	rFlawWaterAfterAlcaliSet:=	arFlawWaterAfterAlcaliSet[3, wChosenRecipeLine3],
	rFlawWaterAfterAccidSet:=	arFlawWaterAfterAccidSet[3, wChosenRecipeLine3],
	rWaterAfterSterilFlaw:=	arWaterAfterSterilFlaw[3, wChosenRecipeLine3],
	rWaterAfterSterilConc:=	arWaterAfterSterilConc[3, wChosenRecipeLine3],
	rFlawWaterAfterAlcaliSet:=	arFlawWaterAfterAlcaliSet[3, wChosenRecipeLine3],
	rFlawWaterAfterAccidSet:=	arFlawWaterAfterAccidSet[3, wChosenRecipeLine3],
	wUsedWaterLevelOK:= wUsedWaterLevelOK,
	wUsedWaterLevelNotOK:= wUsedWaterLevelNotOK,
	wBackTget:= Heater_BackTget_3,
	xPause:= xPauseWashingLine3,
	xVoutOn:= xState_V311,
	xV_NotshortcutOn:= xState_V310,
	xV_UsedWaterInOn:= xState_V308,
	xV_AlkaliInOn:= xState_V306,
	xV_AccidInOn:= xState_V307,
	xV_WaterOutOn:= xState_V301,
	xV_UsedWaterOutOn:= xState_V302,
	xV_AlkaliOutOn:= xState_V304,
	xV_AccidOutOn:= xState_V303,
	xV_CycleOn:= xState_V305,
	xPumpOn:= Pump_OnAuto_3,
	rConcentration:= Conc_Line3,
	(*xAccidIsGoing:=xAccidIsGoing3,*)
	xFeedbackSwitch:= DI_FeedBackSwitchLine3,
	rWaterAfterSterilT:=arWaterAfterSterilT[3, wChosenRecipeLine3],
	wRecipeTimeRinse:= arWaterTime[3, wChosenRecipeLine3],
	wRecipeTimeAlcali:= arAlkaliTime[3, wChosenRecipeLine3],
	wRecipeTimeAccid:= arAccidTime[3, wChosenRecipeLine3],
	wAfterRinseConcAlk:= (*wAfterRinseConcAlk*)rConcSolutionStopoperationAlk,
	wAfterRinseConcAcc:= (*wAfterRinseConcAcc*)rConcSolutionStopoperationAcc,
	wAfterAlkWaterTime:= arAfterAlkaliWaterTime[3, wChosenRecipeLine3],
	wAfterAccWaterTime:= arAfterAccidWaterTime[3, wChosenRecipeLine3],
	rTwaterSet:= arTwaterSet[3, wChosenRecipeLine3],
	rTalcaliSet:= arTalkaliSet[3, wChosenRecipeLine3],
	rTaccidSet:= arTaccidSet[3, wChosenRecipeLine3],
	rConcAlcaliSet:= (*arConcAlkaliSet[3, wChosenRecipeLine3]*)rConcSolutionStartOperationAlk,
	rConcAccidSet:= (*arConcAccidSet[3, wChosenRecipeLine3]*)rConcSolutionStartOperationAcc,
	rFlawAlcaliSet:= arFlawAlkaliSet[3, wChosenRecipeLine3],
	rFlawWaterSet:= arFlawWaterSet[3, wChosenRecipeLine3],
	rFlawAccidSet:= arFlawAccidSet[3, wChosenRecipeLine3],
	wTsteril:= arTsterilSet[3, wChosenRecipeLine3],
	wFlawSteril:= arFlawSterilSet[3, wChosenRecipeLine3],
	rConcSteril:= arConcSterilSet[3, wChosenRecipeLine3],
	wSterilTime:= arSterilTime[3, wChosenRecipeLine3],
	wCountOfOperations:= 7,
	xStart:= xStartWashingLine3,
	xVout:= OnAuto_V311,
	xV_Notshortcut:= OnAuto_V310,
	xV_UsedWaterIn:= OnAuto_V308,
	xV_AlkaliIn:= OnAuto_V306,
	xV_AccidIn:= OnAuto_V307,
	xV_WaterOut:= OnAuto_V301,
	xV_UsedWaterOut:= OnAuto_V302,
	xV_AlkaliOut:= OnAuto_V304,
	xV_AccidOut:= OnAuto_V303,
	xV_Cycle:= OnAuto_V305,
	xV_Drainage:= OnAuto_V309,
	xPump:= Pump_OnAuto_3,
	xHeaterPower:= Heater_AutoSetT_3,
	xResetErrors:= xResetAlmAll,
	xPA:= PA_OnAuto_3,
	rToutSet:= Heater_AutoSetT_3,
	rFlawOutSet:= Pump_FlawAutoSet_3,
	xDone:=xWashingDone_Line3,
	State=> wWashingStateLine3,
	PauseState=>(* wWashingPauseStateLine3*),
	wTimePassed=> wWashingTimePassed3,
	wTimeOperationSet=> wWashingOperTimeSet3,
	wError=> wWashingErr_3);
END_IF
END_PROGRAM

(* POU Process/Washing/prWashingLine4, ST *)
PROGRAM prWashingLine4
VAR
	WashingProcess4:	fbWashingProcess;
	xResetErrors: BOOL;
END_VAR
IF wDissolvingStateLine4 = 0 THEN
WashingProcess4(
	xReady:= (*xReadyForWashing AND*) wDissolvingStateLine4 = 0,
	arOperations:= arOperations,
	rWaterLevel:= CleanWaterLevel,
	rUsedWaterLevel:= UsedWaterLevel,
	rAccidLevel:= AccidLevel,
	rAlkaliLevel:= AlkaliLevel,
	wConcPumpTime:=arConcPumpTimeSteril[4, wChosenRecipeLine4],
	wConcMessureTime:= rConcCheckTime,
	arOperations2x:=arOperations2x,
	arOperations3x:=arOperations3x,
	wChosenRecipeLine:=wChosenRecipeLine4,
	wLine:=4,
	rConcOfClkaliInTank:=rDissolAlkaliConcSet,
	rConcOfAccidInTank:=rDissolAccidConcSet,

	xPumpNorm:=Pump_InvNorm_4,

	rWaterAfterSterilTime:=arWaterAfterSterilTime[4, wChosenRecipeLine4],
	wTafterAlkaliWater:=arTafterAlkaliWater[4, wChosenRecipeLine4],
	wTafterAccidWater:=arTafterAccidWater[4, wChosenRecipeLine4],

	rFlawWaterAfterAlcaliSet:=	arFlawWaterAfterAlcaliSet[4, wChosenRecipeLine4],
	rFlawWaterAfterAccidSet:=	arFlawWaterAfterAccidSet[4, wChosenRecipeLine4],
	rWaterAfterSterilFlaw:=	arWaterAfterSterilFlaw[4, wChosenRecipeLine4],
	rWaterAfterSterilConc:=	arWaterAfterSterilConc[4, wChosenRecipeLine4],
	rFlawWaterAfterAlcaliSet:=	arFlawWaterAfterAlcaliSet[4, wChosenRecipeLine4],
	rFlawWaterAfterAccidSet:=	arFlawWaterAfterAccidSet[4, wChosenRecipeLine4],
	wUsedWaterLevelOK:= wUsedWaterLevelOK,
	wUsedWaterLevelNotOK:= wUsedWaterLevelNotOK,
	wBackTget:= Heater_BackTget_4,
	xPause:= xPauseWashingLine4,
	xVoutOn:= xState_V411,
	xV_NotshortcutOn:= xState_V410,
	xV_UsedWaterInOn:= xState_V408,
	xV_AlkaliInOn:= xState_V406,
	xV_AccidInOn:= xState_V407,
	xV_WaterOutOn:= xState_V401,
	xV_UsedWaterOutOn:= xState_V402,
	xV_AlkaliOutOn:= xState_V404,
	xV_AccidOutOn:= xState_V403,
	xV_CycleOn:= xState_V405,
	xPumpOn:= Pump_OnAuto_4,
	rConcentration:= Conc_Line4,
	(*xAccidIsGoing:=xAccidIsGoing4,*)
	xFeedbackSwitch:= DI_FeedBackSwitchLine4,
	rWaterAfterSterilT:=arWaterAfterSterilT[4, wChosenRecipeLine4],
	wRecipeTimeRinse:= arWaterTime[4, wChosenRecipeLine4],
	wRecipeTimeAlcali:= arAlkaliTime[4, wChosenRecipeLine4],
	wRecipeTimeAccid:= arAccidTime[4, wChosenRecipeLine4],
	wAfterRinseConcAlk:= (*wAfterRinseConcAlk*)rConcSolutionStopoperationAlk,
	wAfterRinseConcAcc:= (*wAfterRinseConcAcc*)rConcSolutionStopoperationAcc,
	wAfterAlkWaterTime:= arAfterAlkaliWaterTime[4, wChosenRecipeLine4],
	wAfterAccWaterTime:= arAfterAccidWaterTime[4, wChosenRecipeLine4],
	rTwaterSet:= arTwaterSet[4, wChosenRecipeLine4],
	rTalcaliSet:= arTalkaliSet[4, wChosenRecipeLine4],
	rTaccidSet:= arTaccidSet[4, wChosenRecipeLine4],
	rConcAlcaliSet:=(* arConcAlkaliSet[4, wChosenRecipeLine4]*)rConcSolutionStartOperationAlk,
	rConcAccidSet:= (*arConcAccidSet[4, wChosenRecipeLine4]*)rConcSolutionStartOperationAcc,
	rFlawAlcaliSet:= arFlawAlkaliSet[4, wChosenRecipeLine4],
	rFlawWaterSet:= arFlawWaterSet[4, wChosenRecipeLine4],
	rFlawAccidSet:= arFlawAccidSet[4, wChosenRecipeLine4],
	wTsteril:= arTsterilSet[4, wChosenRecipeLine4],
	wFlawSteril:= arFlawSterilSet[4, wChosenRecipeLine4],
	rConcSteril:= arConcSterilSet[4, wChosenRecipeLine4],
	wSterilTime:= arSterilTime[4, wChosenRecipeLine4],
	wCountOfOperations:= 7,
	xStart:= xStartWashingLine4,
	xVout:= OnAuto_V411,
	xV_Notshortcut:= OnAuto_V410,
	xV_UsedWaterIn:= OnAuto_V408,
	xV_AlkaliIn:= OnAuto_V406,
	xV_AccidIn:= OnAuto_V407,
	xV_WaterOut:= OnAuto_V401,
	xV_UsedWaterOut:= OnAuto_V402,
	xV_AlkaliOut:= OnAuto_V404,
	xV_AccidOut:= OnAuto_V403,
	xV_Cycle:= OnAuto_V405,
	xV_Drainage:= OnAuto_V409,
	xPump:= Pump_OnAuto_4,
	xHeaterPower:= Heater_AutoSetT_4,
	xResetErrors:= xResetAlmAll,
	xPA:= PA_OnAuto_4,
	rToutSet:= Heater_AutoSetT_4,
	rFlawOutSet:= Pump_FlawAutoSet_4,
	xDone:=xWashingDone_Line4,
	State=> wWashingStateLine4,
	PauseState=> (*wWashingPauseStateLine4*),
	wTimePassed=> wWashingTimePassed4,
	wTimeOperationSet=> wWashingOperTimeSet4,
	wError=> wWashingErr_4);
END_IF
END_PROGRAM

(* POU Simulation_/Simulation, ST *)
PROGRAM Simulation
VAR
	ValveSim_101:fbValveSim;
	ValveSim_102:fbValveSim;
	ValveSim_103:fbValveSim;
	ValveSim_104:fbValveSim;
	ValveSim_105:fbValveSim;
	ValveSim_106:fbValveSim;
	ValveSim_107:fbValveSim;
	ValveSim_108:fbValveSim;
	ValveSim_109:fbValveSim;
	ValveSim_110:fbValveSim;
	ValveSim_111:fbValveSim;
	ValveSim_201:fbValveSim;
	ValveSim_202:fbValveSim;
	ValveSim_203:fbValveSim;
	ValveSim_204:fbValveSim;
	ValveSim_205:fbValveSim;
	ValveSim_206:fbValveSim;
	ValveSim_207:fbValveSim;
	ValveSim_208:fbValveSim;
	ValveSim_209:fbValveSim;
	ValveSim_210:fbValveSim;
	ValveSim_211:fbValveSim;
	ValveSim_301:fbValveSim;
	ValveSim_302:fbValveSim;
	ValveSim_303:fbValveSim;
	ValveSim_304:fbValveSim;
	ValveSim_305:fbValveSim;
	ValveSim_306:fbValveSim;
	ValveSim_307:fbValveSim;
	ValveSim_308:fbValveSim;
	ValveSim_309:fbValveSim;
	ValveSim_310:fbValveSim;
	ValveSim_311:fbValveSim;
	ValveSim_401:fbValveSim;
	ValveSim_402:fbValveSim;
	ValveSim_403:fbValveSim;
	ValveSim_404:fbValveSim;
	ValveSim_405:fbValveSim;
	ValveSim_406:fbValveSim;
	ValveSim_407:fbValveSim;
	ValveSim_408:fbValveSim;
	ValveSim_409:fbValveSim;
	ValveSim_410:fbValveSim;
	ValveSim_411:fbValveSim;
	ValveSim_501:fbValveSim;
	ValveSim_510:fbValveSim;
	ValveSim_511:fbValveSim;
	ValveSim_512:fbValveSim;
	ValveSim_513:fbValveSim;
	ValveSim_514:fbValveSim;
	ValveSim_515:fbValveSim;

	Pump_1:fbValveSim;
	Pump_2:fbValveSim;
	Pump_3:fbValveSim;
	Pump_4:fbValveSim;

END_VAR
ValveSim_101(xDO:= DO_V101, xSensor=> DI_V101);
ValveSim_102(xDO:= DO_V102, xSensor=> DI_V102);
ValveSim_103(xDO:= DO_V103, xSensor=> DI_V103);
ValveSim_104(xDO:= DO_V104, xSensor=> DI_V104);
ValveSim_105(xDO:= DO_V105, xSensor=> DI_V105);
ValveSim_106(xDO:= DO_V106, xSensor=> DI_V106);
ValveSim_107(xDO:= DO_V107, xSensor=> DI_V107);
ValveSim_108(xDO:= DO_V108, xSensor=> DI_V108);
ValveSim_109(xDO:= DO_V109, xSensor=> DI_V109);
ValveSim_110(xDO:= DO_V110, xSensor=> DI_V110);
ValveSim_111(xDO:= DO_V111, xSensor=> DI_V111);
ValveSim_201(xDO:= DO_V201, xSensor=> DI_V201);
ValveSim_202(xDO:= DO_V202, xSensor=> DI_V202);
ValveSim_203(xDO:= DO_V203, xSensor=> DI_V203);
ValveSim_204(xDO:= DO_V204, xSensor=> DI_V204);
ValveSim_205(xDO:= DO_V205, xSensor=> DI_V205);
ValveSim_206(xDO:= DO_V206, xSensor=> DI_V206);
ValveSim_207(xDO:= DO_V207, xSensor=> DI_V207);
ValveSim_208(xDO:= DO_V208, xSensor=> DI_V208);
ValveSim_209(xDO:= DO_V209, xSensor=> DI_V209);
ValveSim_210(xDO:= DO_V210, xSensor=> DI_V210);
ValveSim_211(xDO:= DO_V211, xSensor=> DI_V211);
ValveSim_301(xDO:= DO_V301, xSensor=> DI_V301);
ValveSim_302(xDO:= DO_V302, xSensor=> DI_V302);
ValveSim_303(xDO:= DO_V303, xSensor=> DI_V303);
ValveSim_304(xDO:= DO_V304, xSensor=> DI_V304);
ValveSim_305(xDO:= DO_V305, xSensor=> DI_V305);
ValveSim_306(xDO:= DO_V306, xSensor=> DI_V306);
ValveSim_307(xDO:= DO_V307, xSensor=> DI_V307);
ValveSim_308(xDO:= DO_V308, xSensor=> DI_V308);
ValveSim_309(xDO:= DO_V309, xSensor=> DI_V309);
ValveSim_310(xDO:= DO_V310, xSensor=> DI_V310);
ValveSim_311(xDO:= DO_V311, xSensor=> DI_V311);
ValveSim_401(xDO:= DO_V401, xSensor=> DI_V401);
ValveSim_402(xDO:= DO_V402, xSensor=> DI_V402);
ValveSim_403(xDO:= DO_V403, xSensor=> DI_V403);
ValveSim_404(xDO:= DO_V404, xSensor=> DI_V404);
ValveSim_405(xDO:= DO_V405, xSensor=> DI_V405);
ValveSim_406(xDO:= DO_V406, xSensor=> DI_V406);
ValveSim_407(xDO:= DO_V407, xSensor=> DI_V407);
ValveSim_408(xDO:= DO_V408, xSensor=> DI_V408);
ValveSim_409(xDO:= DO_V409, xSensor=> DI_V409);
ValveSim_410(xDO:= DO_V410, xSensor=> DI_V410);
ValveSim_411(xDO:= DO_V411, xSensor=> DI_V411);
ValveSim_501(xDO:= DO_V501, xSensor=> DI_V501);
ValveSim_510(xDO:= DO_V510, xSensor=> DI_V510);
ValveSim_511(xDO:= DO_V511, xSensor=> DI_V511);
ValveSim_512(xDO:= DO_V512, xSensor=> DI_V512);
ValveSim_513(xDO:= DO_V513, xSensor=> DI_V513);
ValveSim_514(xDO:= DO_V514, xSensor=> DI_V514);
ValveSim_515(xDO:= DO_V515, xSensor=> DI_V515);

Pump_1(xDO:= Pump_OnAuto_1, xSensor=> DI_FeedBackSwitchLine1);
Pump_2(xDO:= Pump_OnAuto_2, xSensor=> DI_FeedBackSwitchLine2);
Pump_3(xDO:= Pump_OnAuto_3, xSensor=> DI_FeedBackSwitchLine3);
Pump_4(xDO:= Pump_OnAuto_4, xSensor=> DI_FeedBackSwitchLine4);
Pump_FeedbackOn_1:=DI_FeedBackSwitchLine1;
Pump_FeedbackOn_2:=DI_FeedBackSwitchLine2;
Pump_FeedbackOn_3:=DI_FeedBackSwitchLine3;
Pump_FeedbackOn_4:=DI_FeedBackSwitchLine4;

Pump_InvNorm_1:=TRUE;
Pump_InvNorm_2:=TRUE;
Pump_InvNorm_3:=TRUE;
Pump_InvNorm_4:=TRUE;
(*
DI_WaterUpperLevel:= FALSE;
DI_UsedWaterUpperLevel:= FALSE;

DI_AlkaliUpperLevel:= FALSE;
DI_AccidUpperLevel:= FALSE;
*)
END_PROGRAM

(* POU Simulation_/fbValveSim, ST *)
FUNCTION_BLOCK fbValveSim
VAR_INPUT
	xDO:	BOOL;
END_VAR
VAR_OUTPUT
	xSensor:	BOOL;
END_VAR
VAR
	tnOn:	TON;
END_VAR
tnOn(IN:=xDO, pt:=t#2s, Q=>xSensor);
END_FUNCTION_BLOCK

(* POU Device/Sensors/fb_counter, ST *)
FUNCTION_BLOCK fb_counter
VAR_INPUT
	repair	:					BOOL	;
	counter	:				BOOL	;
	counter_valueStep	:	REAL	:=	1.0	;
	counter_init_value	:	REAL	;		
	start	:					BOOL	;
END_VAR

VAR_IN_OUT
	reset:			BOOL;
END_VAR

VAR_OUTPUT
	result:						REAL;
END_VAR

VAR
	status_counter:		BOOL;
END_VAR
(*couter di signals*)
IF repair = FALSE
  THEN
    IF start = TRUE
      THEN
        IF status_counter <> counter
          THEN
            IF counter = TRUE
              THEN
                result:= result + counter_valueStep;
            END_IF;
        END_IF;
        status_counter := counter;
    END_IF;

    IF reset = TRUE
      THEN
        reset:= FALSE;
        result:= counter_init_value;
    END_IF;
  ELSE
    result:= 0;
    reset:=FALSE;
    status_counter:= FALSE;
END_IF;
END_FUNCTION_BLOCK

(* POU Device/Sensors/fb_crash_to_int, ST *)
FUNCTION_BLOCK fb_crash_to_int
VAR_INPUT
	repair	:	BOOL	;
	crash_1	:	BOOL	;
	crash_2	:	BOOL	;
	crash_3	:	BOOL	;
	crash_4	:	BOOL	;
	crash_5	:	BOOL	;
	crash_6	:	BOOL	;
	crash_7	:	BOOL	;
	crash_8	:	BOOL	;
	crash_9	:	BOOL	;
	crash_10	:	BOOL	;

END_VAR
VAR_OUTPUT
	rezult_int_crash:	WORD;
END_VAR
VAR
END_VAR
IF repair = FALSE
  THEN
    rezult_int_crash:= INT_TO_WORD(
      (1) * BOOL_TO_INT(crash_1 OR crash_2 OR crash_3 OR crash_4 OR crash_5 OR crash_6 OR crash_7 OR crash_8 OR crash_9 OR crash_10) +
      (2) * BOOL_TO_INT(crash_1) +
      (4) * BOOL_TO_INT(crash_2) +
      (8) * BOOL_TO_INT(crash_3) +
      (16) * BOOL_TO_INT(crash_4) +
      (32) * BOOL_TO_INT(crash_5) +
      (64) * BOOL_TO_INT(crash_6) +
      (128) * BOOL_TO_INT(crash_7) +
      (256) * BOOL_TO_INT(crash_8) +
      (512) * BOOL_TO_INT(crash_9) +
      (1024) * BOOL_TO_INT(crash_10) );
  ELSE
      rezult_int_crash:= 0;
END_IF;
END_FUNCTION_BLOCK

(* POU _ExtraFB/ControlFB/fb_digout_signal, ST *)
FUNCTION_BLOCK fb_digout_signal
VAR_INPUT
	repair	:						BOOL	;
	out_signal_for_repair	:		BOOL	;
	use_smoothing	:			BOOL	;
	time_wait	:					TIME	:=	T#1s500ms	;
	input	:						BOOL	;

END_VAR
VAR_OUTPUT
	digout:							BOOL;
END_VAR
VAR
	perem_input:					BOOL	;
	TON_wait:						TON;
END_VAR
IF repair = FALSE
  THEN
    IF use_smoothing = FALSE
      THEN
        (*???? ?????? ??????????? ????? ?????*)
        digout:= input;
      ELSE
        (*???? ???? ???????? ??????? ?????? ? ?? ?????? ?????????????? ???????? ????????*)
        IF input <> perem_input
          THEN
            TON_wait( IN:=TRUE, PT:= time_wait);
          ELSE
            TON_wait( IN:=FALSE, PT:= time_wait);
        END_IF;
        IF TON_wait.Q = TRUE
          THEN
            digout:= input;
            perem_input:= input;
            TON_wait( IN:=FALSE, PT:= time_wait);
        END_IF;
    END_IF;
  ELSE
    digout:= out_signal_for_repair;
END_IF;
  
END_FUNCTION_BLOCK

(* POU Device/Sensors/fb_speed_di, ST *)
FUNCTION_BLOCK fb_speed_di
VAR_INPUT
	repair	:				BOOL	;
	di_speed	:			BOOL	;
	real_obor_min	:	REAL	:=	1500.0	;
	max_speed	:		REAL	:=	1500.0	;
	time_update	:		DINT	:=	1500	;

END_VAR
VAR_OUTPUT
	result_speed:			REAL;
END_VAR
VAR
	TON_speed	:		TON	;
	status_di_speed	:	BOOL	;
	count_impuls	:		REAL	;

END_VAR
(*translate di speed in speed*)
IF repair = FALSE
  THEN
    IF (status_di_speed = FALSE AND di_speed = TRUE)
      THEN
        count_impuls:= count_impuls + 1;
    END_IF;

    TON_speed( IN:= TRUE, PT:=  DINT_TO_TIME(time_update));
    IF TON_speed.Q = TRUE
      THEN
        TON_speed( IN:= FALSE, PT:=  t#60s);
        IF real_obor_min <> 0 AND time_update <> 0
          THEN
            result_speed:= max_speed * ((count_impuls * 60.0 / (DINT_TO_REAL(time_update) / 1000.0)) / real_obor_min);
          ELSE
            result_speed:= 0;
        END_IF;
        count_impuls:= 0;
    END_IF;

    status_di_speed:= di_speed;
  ELSE
    result_speed:= 0;
    TON_speed( IN:= FALSE, PT:=  t#10d);
    status_di_speed:= FALSE;
    count_impuls:= 0;
END_IF;
END_FUNCTION_BLOCK

(* POU Device/Sensors/fb_tank, ST *)
FUNCTION_BLOCK fb_tank
VAR_INPUT
	use_smoothing	:	BOOL	;
	time_wait	:			TIME	:=	T#1s500ms	;
	input_H	:			BOOL	;
	input_M	:			BOOL	;
	input_L	:			BOOL	;

END_VAR
VAR_OUTPUT
	result_H	:			BOOL	;
	result_M	:			BOOL	;
	result_L	:			BOOL	;
	crash_value	:		BOOL	;
	out_crash_int	:		WORD	;

END_VAR
VAR
	sensor_H	:			fb_digout_signal	;
	sensor_M	:			fb_digout_signal	;
	sensor_L	:			fb_digout_signal	;
	db_crash_to_int	:	fb_crash_to_int	;

END_VAR
(*high level*)
sensor_H(
  repair:=                 FALSE,
  out_signal_for_repair:=  FALSE,
  use_smoothing:=          use_smoothing,
  time_wait:=              time_wait,
  input:=                  input_H,
  digout=>                 result_H);
(*middle level*)
sensor_M(
  repair:=                 FALSE,
  out_signal_for_repair:=  FALSE,
  use_smoothing:=          use_smoothing,
  time_wait:=              time_wait,
  input:=                  input_M,
  digout=>                 result_M);
(*lower level*)
sensor_L(
  repair:=                 FALSE,
  out_signal_for_repair:=  FALSE,
  use_smoothing:=          use_smoothing,
  time_wait:=              time_wait,
  input:=                  input_L,
  digout=>                 result_L);

(*IF (result_M = TRUE AND result_L = FALSE) OR (result_H = TRUE AND result_M = FALSE)
  THEN
    crash_value:= TRUE;
  ELSE
    crash_value:= FALSE;
END_IF;*)
    crash_value:= FALSE;

  
(*?????? ??? ??????*)
db_crash_to_int(
  crash_1:= crash_value );
out_crash_int:= db_crash_to_int.rezult_int_crash;
END_FUNCTION_BLOCK

(* POU Process/SelfWashing/fbWashingTanks, ST *)
FUNCTION_BLOCK fbWashingTanks
VAR_INPUT
	xV_AllInState:					BOOL;
	xV_DrainageState:			BOOL;
	xV_TankInState:				BOOL;
	xV_CleanerOutState:			BOOL;
	xV_PrevCleanerOutState:		BOOL;
	wOperTimeSet:				WORD;
	NextState:							SelfWashingStates;
END_VAR
VAR_IN_OUT

	xV_AllIn:						BOOL;
	xV_Drainage:					BOOL;
	xV_TankIn:						BOOL;
	xV_CleanerOut:				BOOL;
	xV_PrevCleanerOut:			BOOL;
	xPumpOn:						BOOL;
	State:							SelfWashingStates;
END_VAR
VAR_OUTPUT
END_VAR
VAR
	tnWashing:					TON;
	xStartOper:					BOOL;
END_VAR
xV_AllIn:=				TRUE;
xV_Drainage:=		TRUE;
xV_TankIn:=			TRUE;
xV_CleanerOut:=		TRUE;
xV_PrevCleanerOut:=	FALSE;

IF (NOT xV_PrevCleanerOutState) AND xV_AllInState AND xV_DrainageState AND xV_TankInState AND xV_CleanerOutState THEN
	xPumpOn:=TRUE;
	xStartOper:=TRUE;
END_IF

tnWashing(IN:=xStartOper,  PT:= (WORD_TO_TIME(wOperTimeSet))*1000);
IF tnWashing.Q THEN
	tnWashing(IN:=FALSE);
	xStartOper:=FALSE;
	State:= NextState;
END_IF
END_FUNCTION_BLOCK

(* POU Device/Sensors/fnAI_TO_CURRENCY, ST *)
FUNCTION fnAI_TO_CURRENCY : REAL
VAR_INPUT
	AI:	WORD;
END_VAR
VAR
	result:REAL;
END_VAR
result:=(WORD_TO_REAL(AI)/32762)*20;
fnAI_TO_CURRENCY:=result;
END_FUNCTION

(* POU Device/Sensors/fnPressureToVolume, ST *)
FUNCTION fnPressureToVolume : REAL
VAR_INPUT
	Pressure:	REAL;
	Square:	REAL;
END_VAR
VAR
END_VAR
fnPressureToVolume:=(Pressure*Square)/9.79038;
END_FUNCTION

(* Visualisation PLC_VISU
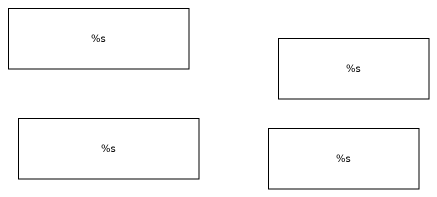
rectangle at (190,130)-(371,191): text "%s"; shows .Heater_Ki; editable
rectangle at (200,240)-(381,301): text "%s"; shows .Heater_Kd; editable
rectangle at (460,160)-(611,221): text "%s"; shows .Pump_Kp; editable
rectangle at (450,250)-(601,311): text "%s"; shows .Pump_Ki; editable
*)
